{attribute 'qualified_only'}
VAR_GLOBAL
	ConveyerAxis 			: AXIS_REF;
	bConveyerReadyToMove 	: BOOL;
	bConveyerReadyToPick 	: BOOL;
	bSensor 				: BOOL;
END_VAR

(* stored: Version 1.1.0.1, ProductVersion 3.1.4024.11
   GVL GVL_Conveyer: Id {4b8a48cf-6d3b-4a7a-9cb1-ab1cbec33255} *)
